// TIA Portal V19 export
TYPE "LAF_typeRollerEm1ProcessValues"
// stored: Access Published
   STRUCT
      pieceCount : DInt;
   END_STRUCT;
END_TYPE
